// TIA Portal V21 export
FUNCTION "FC_Cargador" : Void   // FC3, LAD
TITLE = Sistema de carga de pallets para clasificacion
{ S7_Optimized_Access := 'TRUE' }
// stored: SetENOAutomatically false
   VAR_INPUT
      Loaded : Bool;
      "Sistema en marcha" : Bool;
      Emergencia : Bool;
      "Caja alta" : Bool;
      "Caja baja" : Bool;
      Clasificando : Bool;
   END_VAR
   VAR_OUTPUT
      Load : Bool;
      "Transfer left" : Bool;
      "Transfer right" : Bool;
   END_VAR
BEGIN

REGION Network 1: Activar/Desactivar cinta para acercamiento de pallets a sensor
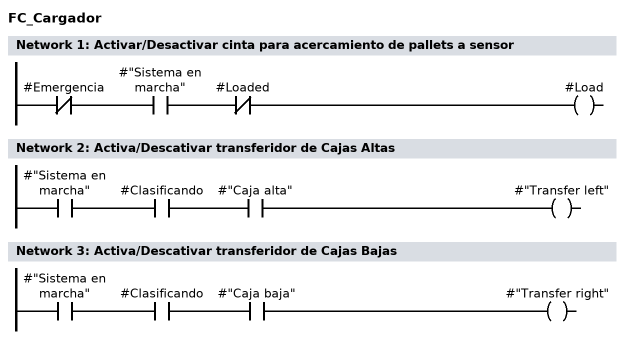
   RUNG wire#powerrail
      I_Contact( #Emergencia )
      Contact( #"Sistema en marcha" )
      I_Contact( #Loaded )
      Coil( #Load )
   END_RUNG
   // the same network as SCL:
   #Load := NOT #Emergencia AND #"Sistema en marcha" AND NOT #Loaded;
END_REGION

REGION Network 2: Activa/Descativar transferidor de Cajas Altas
   RUNG wire#powerrail
      Contact( #"Sistema en marcha" )
      Contact( #Clasificando )
      Contact( #"Caja alta" )
      Coil( #"Transfer left" )
   END_RUNG
   // the same network as SCL:
   #"Transfer left" := #"Sistema en marcha" AND #Clasificando AND #"Caja alta";
END_REGION

REGION Network 3: Activa/Descativar transferidor de Cajas Bajas
   RUNG wire#powerrail
      Contact( #"Sistema en marcha" )
      Contact( #Clasificando )
      Contact( #"Caja baja" )
      Coil( #"Transfer right" )
   END_RUNG
   // the same network as SCL:
   #"Transfer right" := #"Sistema en marcha" AND #Clasificando AND #"Caja baja";
END_REGION
END_FUNCTION
